(* IEC 61131-3 sources: AXOpen/src/components.keyence.vision/ctrl/src (part 3) *)

                    CompletionClearControl.TuneCompleteClear := CompletionStatus.TuneComplete;
                    IF NOT CompletionStatus.TuneComplete THEN
                        CompletionClearControl.TuneCompleteClear := FALSE;
                        THIS.CallTimers(FALSE);
                        _progress := 406;
                    END_IF;
                END_IF;

                IF _progress = 406 THEN             // TuneTask running, clear external request complete flag
                    IF _infoTimer.output THEN
                        TaskMessenger.Activate( UINT#606, eAxoMessageCategory#Warning);
                        Status.Error.Id :=      UINT#606;
                    END_IF;

                    CompletionClearControl.EXT_RequestCompleteClear := CompletionStatus.EXT_RequestComplete;
                    IF NOT CompletionStatus.EXT_RequestComplete THEN
                        CompletionClearControl.EXT_RequestCompleteClear := FALSE;
                        THIS.CallTimers(FALSE);
                        _progress := 407;
                    END_IF;
                END_IF;

                IF _progress = 407 THEN             // TuneTask running, waiting for general error flag is reseted
                    IF _infoTimer.output THEN
                        TaskMessenger.Activate( UINT#607, eAxoMessageCategory#Warning);
                        Status.Error.Id :=      UINT#607;
                    END_IF;

                    IF NOT HandshakeAndGeneralErrorStatus.GeneralError THEN
                        THIS.CallTimers(FALSE);
                        _progress := 408;
                    END_IF;
                END_IF;

                IF _progress = 408 THEN             // TuneTask running, setting bank number
                    IF _infoTimer.output THEN
                        TaskMessenger.Activate( UINT#608, eAxoMessageCategory#Warning);
                        Status.Error.Id :=      UINT#608;
                    END_IF;

                    IF _Bank>=UINT#0 AND _Bank <=UINT#10 THEN
                        ParameterBankNumber.BankNumberRegister := _Bank;
                        THIS.CallTimers(FALSE);
                        _progress := 409;
                    END_IF;
                END_IF;

                IF _progress = 409 THEN             // TuneTask running, starting tune process
                    IF _infoTimer.output THEN
                        TaskMessenger.Activate( UINT#609, eAxoMessageCategory#Warning);
                        Status.Error.Id :=      UINT#609;
                    END_IF;

                    OperationInstructionControl.TuneRequest := TRUE;
                    IF CompletionStatus.TuneComplete THEN
                        OperationInstructionControl.TuneRequest := FALSE;
                        THIS.CallTimers(FALSE);
                        IF NOT ErrorStatus.TuneFailure THEN
                            _progress := 410;
                        ELSE
                            TuneTask.ThrowWhen(TRUE,'ErrorStatus.TuneFailure');
                        END_IF;
                    END_IF;
                END_IF;

                IF _progress = 410 THEN             // TuneTask running, acknowledging tunning process
                    IF _infoTimer.output THEN
                        TaskMessenger.Activate( UINT#610, eAxoMessageCategory#Warning);
                        Status.Error.Id :=      UINT#610;
                    END_IF;

                    CompletionClearControl.TuneCompleteClear := TRUE;
                    IF NOT CompletionStatus.TuneComplete THEN
                        CompletionClearControl.TuneCompleteClear := FALSE;
                        _progress := 411;
                    END_IF;
                END_IF;

                IF _progress = 411 THEN             // TuneTask running,
                    IF _infoTimer.output THEN
                        TaskMessenger.Activate( UINT#611, eAxoMessageCategory#Warning);
                        Status.Error.Id :=      UINT#611;
                    END_IF;

                    IF TRUE THEN
                        _progress := 412;
                    END_IF;
                END_IF;

                IF _progress = 412 THEN             // TuneTask running,
                    IF _infoTimer.output THEN
                        TaskMessenger.Activate( UINT#612, eAxoMessageCategory#Warning);
                        Status.Error.Id :=      UINT#612;
                    END_IF;

                    IF TRUE THEN
                        _progress := 413;
                    END_IF;
                END_IF;

                IF _progress = 413 THEN             // TuneTask running,
                    IF _infoTimer.output THEN
                        TaskMessenger.Activate( UINT#613, eAxoMessageCategory#Warning);
                        Status.Error.Id :=      UINT#613;
                    END_IF;

                    IF TRUE THEN
                        _progress := 414;
                    END_IF;
                END_IF;

                IF _progress = 414 THEN             // TuneTask running,
                    IF _infoTimer.output THEN
                        TaskMessenger.Activate( UINT#614, eAxoMessageCategory#Warning);
                        Status.Error.Id :=      UINT#614;
                    END_IF;

                    IF TRUE THEN
                        _progress := 415;
                    END_IF;
                END_IF;

                IF _progress = 415 THEN             // TuneTask running,
                    IF _infoTimer.output THEN
                        TaskMessenger.Activate( UINT#615, eAxoMessageCategory#Warning);
                        Status.Error.Id :=      UINT#615;
                    END_IF;

                    IF TRUE THEN
                        _progress := 416;
                    END_IF;
                END_IF;

                IF _progress = 416 THEN             // TuneTask running,
                    IF _infoTimer.output THEN
                        TaskMessenger.Activate( UINT#616, eAxoMessageCategory#Warning);
                        Status.Error.Id :=      UINT#616;
                    END_IF;

                    IF TRUE THEN
                        _progress := 417;
                    END_IF;
                END_IF;

                IF _progress = 417 THEN             // TuneTask running,
                    IF _infoTimer.output THEN
                        TaskMessenger.Activate( UINT#617, eAxoMessageCategory#Warning);
                        Status.Error.Id :=      UINT#617;
                    END_IF;

                    IF TRUE THEN
                        _progress := 418;
                    END_IF;
                END_IF;

                IF _progress = 418 THEN             // TuneTask running,
                    IF _infoTimer.output THEN
                        TaskMessenger.Activate( UINT#618, eAxoMessageCategory#Warning);
                        Status.Error.Id :=      UINT#618;
                    END_IF;

                    IF TRUE THEN
                        _progress := 419;
                    END_IF;
                END_IF;

                IF _progress = 419 THEN             // TuneTask finished
                    TuneTask.DoneWhen(TRUE);
                    _progress := 0;
                END_IF;

                THIS.CallTimers(TRUE);

                TuneTask.ThrowWhen(_errorTimer.output);
                Status.Action.Id := TO_UINT(_progress);
            END_IF;
            IF TuneTask.DoneReached() THEN
                Status.Action.Id :=  UINT#201;
                Status.Error.Id :=  UINT#0;
            ELSIF TuneTask.ErrorOccured() THEN
                Status.Action.Id :=  UINT#10100;
                Status.Error.Id  :=  UINT#10100;
            ELSIF TuneTask.AbortTriggered()THEN
                Status.Action.Id :=  UINT#10101;
                Status.Error.Id  :=  UINT#10101;
            END_IF;
            Messenger.ActivateOnCondition(ULINT#10100,TuneTask.HasError(), eAxoMessageCategory#Error);
            Messenger.ActivateOnCondition(ULINT#10101,TuneTask.IsAborted(), eAxoMessageCategory#Error);
            Messenger.ActivateOnCondition(ULINT#202,TuneTask.RestoreTriggered() , eAxoMessageCategory#Error);
            IF TuneTask.RestoreTriggered() AND _progress >= 400 AND _progress <= 419  THEN
                Status.Action.Id :=  UINT#202;
                _progress := 0;
            END_IF;
            //******************************************

            //****************Update outputs*****************
            _data_1[0].%X1                  :=      LatchAndErrorClearControl.ResultDataLatch;
            _data_1[0].%X7                  :=      LatchAndErrorClearControl.ErrorClear;

            _retVal := Siemens.Simatic.S71500.DistributedIO.WriteData(_hwIdLatchAndErrorClearControl,_data_1);
            IF _retVal > WORD#0 THEN
                Messenger.Activate(UINT#1231, eAxoMessageCategory#ProgrammingError);
                Status.Error.Id := UINT#1231;
                RETURN;
            END_IF;

            _data_1[0].%X0                  :=      OperationInstructionControl.ReadRequest;
            _data_1[0].%X1                  :=      OperationInstructionControl.PresetRequest;
            _data_1[0].%X2                  :=      OperationInstructionControl.RegisterPresetDataRequest;
            _data_1[0].%X3                  :=      OperationInstructionControl.TuneRequest;

            _retVal := Siemens.Simatic.S71500.DistributedIO.WriteData(_hwIdOperationInstructionControl,_data_1);
            IF _retVal > WORD#0 THEN
                Messenger.Activate(UINT#1232, eAxoMessageCategory#ProgrammingError);
                Status.Error.Id := UINT#1232;
                RETURN;
            END_IF;

            _data_1[0].%X0                  :=      CompletionClearControl.ReadCompleteClear;
            _data_1[0].%X1                  :=      CompletionClearControl.PresetCompleteClear;
            _data_1[0].%X2                  :=      CompletionClearControl.RegisterPresetDataCompleteClear;
            _data_1[0].%X3                  :=      CompletionClearControl.TuneCompleteClear;
            _data_1[0].%X7                  :=      CompletionClearControl.EXT_RequestCompleteClear;

            _retVal := Siemens.Simatic.S71500.DistributedIO.WriteData(_hwIdCompletionClearControl,_data_1);
            IF _retVal > WORD#0 THEN
                Messenger.Activate(UINT#1233, eAxoMessageCategory#ProgrammingError);
                Status.Error.Id := UINT#1233;
                RETURN;
            END_IF;

            _data_2[1]                      :=      TO_WORD(ParameterBankNumber.BankNumberRegister).%B0;
            _data_2[0]                      :=      TO_WORD(ParameterBankNumber.BankNumberRegister).%B1;

            _retVal := Siemens.Simatic.S71500.DistributedIO.WriteData(_hwIdParameterBankNumber,_data_2);
            IF _retVal > WORD#0 THEN
                Messenger.Activate(UINT#1234, eAxoMessageCategory#ProgrammingError);
                Status.Error.Id := UINT#1234;
                RETURN;
            END_IF;

            _invalidDataSize := NOT ( Config.UserDataSize = eAxo_SR_750_UserDataSize#USER_DATA_32B OR
                                      Config.UserDataSize = eAxo_SR_750_UserDataSize#USER_DATA_64B OR
                                      Config.UserDataSize = eAxo_SR_750_UserDataSize#USER_DATA_128B OR
                                      Config.UserDataSize = eAxo_SR_750_UserDataSize#USER_DATA_252B);

            IF _invalidDataSize THEN
                Messenger.Activate(UINT#1235, eAxoMessageCategory#ProgrammingError);
                Status.Error.Id := UINT#1235;
                RETURN;
            END_IF;

            IF (UserData.DataChanged <> _UserDataChanged) THEN
                IF Config.UserDataSize = eAxo_SR_750_UserDataSize#USER_DATA_32B THEN
                    _data_34[1] := TO_WORD(User.UserDataSize).%B0;
                    _data_34[0] := TO_WORD(User.UserDataSize).%B1;
                    FOR _index := 2 TO 33 DO
                        _data_34[_index] := UserData.Data[_index];
                    END_FOR;
                    _retVal := Siemens.Simatic.S71500.DistributedIO.WriteData(_hwIdUserData ,_data_34);
                    IF _retVal > WORD#0 THEN
                        Messenger.Activate(UINT#1236, eAxoMessageCategory#ProgrammingError);
                        Status.Error.Id := UINT#1236;
                        RETURN;
                    END_IF;
                ELSIF Config.UserDataSize = eAxo_SR_750_UserDataSize#USER_DATA_64B THEN
                    _data_66[1] := TO_WORD(User.UserDataSize).%B0;
                    _data_66[0] := TO_WORD(User.UserDataSize).%B1;
                    FOR _index := 2 TO 65 DO
                        _data_66[_index] := UserData.Data[_index];
                    END_FOR;
                    _retVal := Siemens.Simatic.S71500.DistributedIO.WriteData(_hwIdUserData ,_data_66);
                    IF _retVal > WORD#0 THEN
                        Messenger.Activate(UINT#1237, eAxoMessageCategory#ProgrammingError);
                        Status.Error.Id := UINT#1237;
                        RETURN;
                    END_IF;
                ELSIF Config.UserDataSize = eAxo_SR_750_UserDataSize#USER_DATA_128B THEN
                    _data_130[1] := TO_WORD(User.UserDataSize).%B0;
                    _data_130[0] := TO_WORD(User.UserDataSize).%B1;
                    FOR _index := 2 TO 129 DO
                        _data_130[_index] := UserData.Data[_index];
                    END_FOR;
                    _retVal := Siemens.Simatic.S71500.DistributedIO.WriteData(_hwIdUserData ,_data_130);
                    IF _retVal > WORD#0 THEN
                        Messenger.Activate(UINT#1238, eAxoMessageCategory#ProgrammingError);
                        Status.Error.Id := UINT#1238;
                        RETURN;
                    END_IF;
                ELSIF Config.UserDataSize = eAxo_SR_750_UserDataSize#USER_DATA_252B THEN
                    _data_254[1] := TO_WORD(User.UserDataSize).%B0;
                    _data_254[0] := TO_WORD(User.UserDataSize).%B1;
                    FOR _index := 2 TO 253 DO
                        _data_254[_index] := UserData.Data[_index];
                    END_FOR;
                    _retVal := Siemens.Simatic.S71500.DistributedIO.WriteData(_hwIdUserData ,_data_254);
                    IF _retVal > WORD#0 THEN
                        Messenger.Activate(UINT#1239, eAxoMessageCategory#ProgrammingError);
                        Status.Error.Id := UINT#1239;
                        RETURN;
                    END_IF;
                END_IF;
                _UserDataChanged := UserData.DataChanged;
            END_IF;
        END_METHOD

        ///<summary>
		/// Clears the result data.
        ///</summary>
        METHOD PUBLIC ClearResultData : IAxoTaskState
            ClearResultData :=ClearResultDataTask.Invoke(THIS);;
        END_METHOD

        ///<summary>
		/// Triggers the reading sequence and waits for results.
        ///</summary>
        METHOD PUBLIC Read : IAxoTaskState
            VAR_INPUT
                inBank : UINT;
            END_VAR
            VAR_OUTPUT
                result : ARRAY [0..245] OF BYTE;
            END_VAR
            _Bank := inBank;
            result := ResultData.Data;
            Read := ReadTask.Invoke(THIS);
        END_METHOD

        ///<summary>
		/// Triggers the reading sequence and waits for results.
        ///</summary>
        METHOD PUBLIC Tune : IAxoTaskState
            VAR_INPUT
                inBank : UINT;
            END_VAR
            _Bank := inBank;
            Tune := TuneTask.Invoke(THIS);
        END_METHOD

        ///<summary>
		/// Triggers the reading sequence and waits for results.
        ///</summary>
        METHOD PUBLIC Read : IAxoTaskState
            VAR_OUTPUT
                result : ARRAY [0..245] OF BYTE;
            END_VAR
            _Bank := UINT#0;
            result := ResultData.Data;
            Read := ReadTask.Invoke(THIS);
        END_METHOD

        METHOD PRIVATE CallTimers
            VAR_INPUT
                signal : BOOL;
            END_VAR

            _infoTimer.OnDelay(THIS, signal , Config.InfoTime);
            _errorTimer.OnDelay(THIS, signal , Config.ErrorTime );
        END_METHOD

        METHOD PRIVATE ContinuousReading //TODO
            VAR
                _index : INT;
            END_VAR
            // IF ResultsStatus.ResultsAvailable AND NOT ResultsControl.ResultsAcknowledge AND Results.Code > UINT#0 AND Results.Length > UINT#0 THEN
            //     Messenger.ActivateOnCondition(ULINT#820, Results.Length > TO_UINT(Config.ResultDataSize), eAxoMessageCategory#Error);
            //     TaskMessenger.ActivateOnCondition(ULINT#713, Results.Length > TO_UINT(Config.ResultDataSize), eAxoMessageCategory#Error);
            //     IF Results.Length > TO_UINT(Config.ResultDataSize) THEN
            //         Status.Action.Id := UINT#820;
            //         Status.Error.Id := UINT#713;
            //     ELSE
            //         FOR _index := 0 TO (TO_INT(Results.Length) - INT#1) DO
            //             ResultData.Data[_index] := _data_in[_index + 8];
            //         END_FOR;
            //         FOR _index := TO_INT(Results.Length) TO 245 DO
            //             ResultData.Data[_index] := BYTE#0;
            //         END_FOR;
            //         ResultData.DataChanged := NOT ResultData.DataChanged ;
            //         Status.Action.Id := UINT#120;
            //     END_IF;
            // END_IF;

            // ResultsControl.ResultsAcknowledge := ResultsStatus.ResultsAvailable;
            ;
        END_METHOD

        ///<summary>
		/// Custom logic for the manual control.
        ///</summary>
        METHOD PROTECTED OVERRIDE ManualControl
            ;
        END_METHOD

        ///<summary>
		/// Restores this instance to its initial state.
        ///</summary>
        METHOD PUBLIC OVERRIDE Restore
            VAR
                _index : INT;
            END_VAR
            Status.Action.Id := UINT#0;
            Status.Error.Id  := UINT#0;
            Messenger.Restore();
            TaskMessenger.Restore();

            ClearResultDataTask.Restore();
            ReadTask.Restore();
            TuneTask.Restore();

            LatchAndErrorClearControl.ResultDataLatch               :=  FALSE;
            LatchAndErrorClearControl.ErrorClear                    :=  FALSE;
            OperationInstructionControl.ReadRequest                 :=  FALSE;
            OperationInstructionControl.PresetRequest               :=  FALSE;
            OperationInstructionControl.RegisterPresetDataRequest	:=  FALSE;
            OperationInstructionControl.TuneRequest	                :=  FALSE;
            CompletionClearControl.ReadCompleteClear	            :=  FALSE;
            CompletionClearControl.PresetCompleteClear	            :=  FALSE;
            CompletionClearControl.RegisterPresetDataCompleteClear	:=  FALSE;
            CompletionClearControl.TuneCompleteClear	            :=  FALSE;
            CompletionClearControl.EXT_RequestCompleteClear	        :=  FALSE;
            ParameterBankNumber.BankNumberRegister	                :=  UINT#0;
            User.UserDataSize                                       :=  UINT#0;

            _prevResultDataReadyCount                               :=  UINT#0;
            _prevResultDataUpdateCount                              :=  UINT#0;
            _resultString                                           :=  '';
            ReadData.ResultDataSize                                 :=  UINT#0;

            FOR _index := 0 TO 245 DO
                ResultData.Data[_index] := BYTE#0;
            END_FOR;

            IF NOT HandshakeAndGeneralErrorStatus.GeneralError THEN
                Status.Action.Id := UINT#50;
                RestoreTask.DoneWhen(TRUE);
            END_IF;
        END_METHOD
    END_CLASS
END_NAMESPACE
